FUNCTION_BLOCK Test_TStreamAdd_Read_BYTE EXTENDS T_UnitTestBase
VAR
    Stream  : T_Stream(StreamLength := 2);
    ArgType : E_ArgTypeId := E_ArgTypeId.Type_BYTE;
END_VAR

Stream.Init(2);

// add a byte...
Stream.SetNextArgTypeId(ArgType);
Stream.Add_BYTE(123);

Stream.SetReadPosition(0);

// check next arg type is correct...
Assertion.AssertEquals_INT(Expected     := ArgType,
                           Actual       := Stream.GetNextArgTypeId(),
                           VariableName := 'Stream.GetNextArgTypeId()');

// check next value...	
Assertion.AssertEquals_BYTE(Expected     := 123,
                            Actual       := Stream.Read_BYTE(),
                            VariableName := 'Stream.Read_BYTE()');

// check we are at the end of the stream..							
Assertion.AssertEquals_UDINT(Expected     := Stream.StreamLength,
                             Actual       := Stream.ReadPosition,
                             VariableName := 'Stream.ReadPosition');

TestFinished();

END_FUNCTION_BLOCK

(* stored: Version 1.1.0.1, ProductVersion 3.1.4024.9
   POU Test_TStreamAdd_Read_BYTE: Id {e2f83219-ac36-4c11-a18b-54f10c7081f6}, SpecialFunc None *)
